# EPICS autosave request: keysight33500B/keysight33500Bchan_settings.req
$(P)$(Q):CH$(CHAN):AMP:TWV
$(P)$(Q):CH$(CHAN):OFF:TWV
$(P)$(Q):CH$(CHAN):UPDATE.SCAN
